//--- Generated by OneClick Automation SourceGenerator v.3.0 ---
DATA_BLOCK DB111
TITLE =Sensors 4-20
AUTHOR:  Kratovi4
VERSION : 2.0
STRUCT
SNS: ARRAY  [1 .. 25] OF
"SNS"; // Array
END_STRUCT ;
BEGIN
END_DATA_BLOCK


DATA_BLOCK DB121
TITLE =Sensors 4-20
AUTHOR:  Kratovi4
VERSION : 2.0
STRUCT
SNS: ARRAY  [1 .. 30] OF
"SNS"; // Array
END_STRUCT ;
BEGIN
END_DATA_BLOCK


DATA_BLOCK DB131
TITLE =Sensors 4-20
AUTHOR:  Kratovi4
VERSION : 2.0
STRUCT
SNS: ARRAY  [1 .. 5] OF
"SNS"; // Array
END_STRUCT ;
BEGIN
END_DATA_BLOCK


DATA_BLOCK DB141
TITLE =Sensors 4-20
AUTHOR:  Kratovi4
VERSION : 2.0
STRUCT
SNS: ARRAY  [1 .. 5] OF
"SNS"; // Array
END_STRUCT ;
BEGIN
END_DATA_BLOCK


DATA_BLOCK DB151
TITLE =Sensors 4-20
AUTHOR:  Kratovi4
VERSION : 2.0
STRUCT
SNS: ARRAY  [1 .. 5] OF
"SNS"; // Array
END_STRUCT ;
BEGIN
END_DATA_BLOCK


DATA_BLOCK DB161
TITLE =Sensors 4-20
AUTHOR:  Kratovi4
VERSION : 2.0
STRUCT
SNS: ARRAY  [1 .. 5] OF
"SNS"; // Array
END_STRUCT ;
BEGIN
END_DATA_BLOCK


DATA_BLOCK DB171
TITLE =Sensors 4-20
AUTHOR:  Kratovi4
VERSION : 2.0
STRUCT
SNS: ARRAY  [1 .. 5] OF
"SNS"; // Array
END_STRUCT ;
BEGIN
END_DATA_BLOCK


DATA_BLOCK DB211
TITLE =Sensors 4-20
AUTHOR:  Kratovi4
VERSION : 2.0
STRUCT
SNS: ARRAY  [1 .. 10] OF
"SNS"; // Array
END_STRUCT ;
BEGIN
END_DATA_BLOCK


DATA_BLOCK DB221
TITLE =Sensors 4-20
AUTHOR:  Kratovi4
VERSION : 2.0
STRUCT
SNS: ARRAY  [1 .. 10] OF
"SNS"; // Array
END_STRUCT ;
BEGIN
END_DATA_BLOCK


DATA_BLOCK DB231
TITLE =Sensors 4-20
AUTHOR:  Kratovi4
VERSION : 2.0
STRUCT
SNS: ARRAY  [1 .. 10] OF
"SNS"; // Array
END_STRUCT ;
BEGIN
END_DATA_BLOCK


DATA_BLOCK DB241
TITLE =Sensors 4-20
AUTHOR:  Kratovi4
VERSION : 2.0
STRUCT
SNS: ARRAY  [1 .. 5] OF
"SNS"; // Array
END_STRUCT ;
BEGIN
END_DATA_BLOCK


DATA_BLOCK DB251
TITLE =Sensors 4-20
AUTHOR:  Kratovi4
VERSION : 2.0
STRUCT
SNS: ARRAY  [1 .. 5] OF
"SNS"; // Array
END_STRUCT ;
BEGIN
END_DATA_BLOCK


DATA_BLOCK DB261
TITLE =Sensors 4-20
AUTHOR:  Kratovi4
VERSION : 2.0
STRUCT
SNS: ARRAY  [1 .. 5] OF
"SNS"; // Array
END_STRUCT ;
BEGIN
END_DATA_BLOCK


DATA_BLOCK DB291
TITLE =Sensors 4-20
AUTHOR:  Kratovi4
VERSION : 2.0
STRUCT
SNS: ARRAY  [1 .. 25] OF
"SNS"; // Array
END_STRUCT ;
BEGIN
END_DATA_BLOCK


DATA_BLOCK DB301
TITLE =Sensors 4-20
AUTHOR:  Kratovi4
VERSION : 2.0
STRUCT
SNS: ARRAY  [1 .. 10] OF
"SNS"; // Array
END_STRUCT ;
BEGIN
END_DATA_BLOCK


DATA_BLOCK DB311
TITLE =Sensors 4-20
AUTHOR:  Kratovi4
VERSION : 2.0
STRUCT
SNS: ARRAY  [1 .. 5] OF
"SNS"; // Array
END_STRUCT ;
BEGIN
END_DATA_BLOCK


DATA_BLOCK DB321
TITLE =Sensors 4-20
AUTHOR:  Kratovi4
VERSION : 2.0
STRUCT
SNS: ARRAY  [1 .. 5] OF
"SNS"; // Array
END_STRUCT ;
BEGIN
END_DATA_BLOCK


DATA_BLOCK DB341
TITLE =Sensors 4-20
AUTHOR:  Kratovi4
VERSION : 2.0
STRUCT
SNS: ARRAY  [1 .. 5] OF
"SNS"; // Array
END_STRUCT ;
BEGIN
END_DATA_BLOCK


DATA_BLOCK DB431
TITLE =Sensors 4-20
AUTHOR:  Kratovi4
VERSION : 2.0
STRUCT
SNS: ARRAY  [1 .. 20] OF
"SNS"; // Array
END_STRUCT ;
BEGIN
END_DATA_BLOCK


DATA_BLOCK DB441
TITLE =Sensors 4-20
AUTHOR:  Kratovi4
VERSION : 2.0
STRUCT
SNS: ARRAY  [1 .. 5] OF
"SNS"; // Array
END_STRUCT ;
BEGIN
END_DATA_BLOCK


DATA_BLOCK DB451
TITLE =Sensors 4-20
AUTHOR:  Kratovi4
VERSION : 2.0
STRUCT
SNS: ARRAY  [1 .. 5] OF
"SNS"; // Array
END_STRUCT ;
BEGIN
END_DATA_BLOCK


DATA_BLOCK DB461
TITLE =Sensors 4-20
AUTHOR:  Kratovi4
VERSION : 2.0
STRUCT
SNS: ARRAY  [1 .. 5] OF
"SNS"; // Array
END_STRUCT ;
BEGIN
END_DATA_BLOCK


DATA_BLOCK DB471
TITLE =Sensors 4-20
AUTHOR:  Kratovi4
VERSION : 2.0
STRUCT
SNS: ARRAY  [1 .. 5] OF
"SNS"; // Array
END_STRUCT ;
BEGIN
END_DATA_BLOCK


DATA_BLOCK DB511
TITLE =Sensors 4-20
AUTHOR:  Kratovi4
VERSION : 2.0
STRUCT
SNS: ARRAY  [1 .. 5] OF
"SNS"; // Array
END_STRUCT ;
BEGIN
END_DATA_BLOCK


DATA_BLOCK DB521
TITLE =Sensors 4-20
AUTHOR:  Kratovi4
VERSION : 2.0
STRUCT
SNS: ARRAY  [1 .. 5] OF
"SNS"; // Array
END_STRUCT ;
BEGIN
END_DATA_BLOCK


DATA_BLOCK DB531
TITLE =Sensors 4-20
AUTHOR:  Kratovi4
VERSION : 2.0
STRUCT
SNS: ARRAY  [1 .. 5] OF
"SNS"; // Array
END_STRUCT ;
BEGIN
END_DATA_BLOCK


DATA_BLOCK DB541
TITLE =Sensors 4-20
AUTHOR:  Kratovi4
VERSION : 2.0
STRUCT
SNS: ARRAY  [1 .. 5] OF
"SNS"; // Array
END_STRUCT ;
BEGIN
END_DATA_BLOCK


DATA_BLOCK DB561
TITLE =Sensors 4-20
AUTHOR:  Kratovi4
VERSION : 2.0
STRUCT
SNS: ARRAY  [1 .. 5] OF
"SNS"; // Array
END_STRUCT ;
BEGIN
END_DATA_BLOCK


DATA_BLOCK DB571
TITLE =Sensors 4-20
AUTHOR:  Kratovi4
VERSION : 2.0
STRUCT
SNS: ARRAY  [1 .. 5] OF
"SNS"; // Array
END_STRUCT ;
BEGIN
END_DATA_BLOCK


DATA_BLOCK DB581
TITLE =Sensors 4-20
AUTHOR:  Kratovi4
VERSION : 2.0
STRUCT
SNS: ARRAY  [1 .. 5] OF
"SNS"; // Array
END_STRUCT ;
BEGIN
END_DATA_BLOCK


DATA_BLOCK DB611
TITLE =Sensors 4-20
AUTHOR:  Kratovi4
VERSION : 2.0
STRUCT
SNS: ARRAY  [1 .. 5] OF
"SNS"; // Array
END_STRUCT ;
BEGIN
END_DATA_BLOCK


DATA_BLOCK DB671
TITLE =Sensors 4-20
AUTHOR:  Kratovi4
VERSION : 2.0
STRUCT
SNS: ARRAY  [1 .. 10] OF
"SNS"; // Array
END_STRUCT ;
BEGIN
END_DATA_BLOCK


DATA_BLOCK DB681
TITLE =Sensors 4-20
AUTHOR:  Kratovi4
VERSION : 2.0
STRUCT
SNS: ARRAY  [1 .. 5] OF
"SNS"; // Array
END_STRUCT ;
BEGIN
END_DATA_BLOCK


DATA_BLOCK DB691
TITLE =Sensors 4-20
AUTHOR:  Kratovi4
VERSION : 2.0
STRUCT
SNS: ARRAY  [1 .. 5] OF
"SNS"; // Array
END_STRUCT ;
BEGIN
END_DATA_BLOCK


DATA_BLOCK DB701
TITLE =Sensors 4-20
AUTHOR:  Kratovi4
VERSION : 2.0
STRUCT
SNS: ARRAY  [1 .. 5] OF
"SNS"; // Array
END_STRUCT ;
BEGIN
END_DATA_BLOCK


DATA_BLOCK DB711
TITLE =Sensors 4-20
AUTHOR:  Kratovi4
VERSION : 2.0
STRUCT
SNS: ARRAY  [1 .. 5] OF
"SNS"; // Array
END_STRUCT ;
BEGIN
END_DATA_BLOCK


DATA_BLOCK DB721
TITLE =Sensors 4-20
AUTHOR:  Kratovi4
VERSION : 2.0
STRUCT
SNS: ARRAY  [1 .. 15] OF
"SNS"; // Array
END_STRUCT ;
BEGIN
END_DATA_BLOCK


DATA_BLOCK DB731
TITLE =Sensors 4-20
AUTHOR:  Kratovi4
VERSION : 2.0
STRUCT
SNS: ARRAY  [1 .. 5] OF
"SNS"; // Array
END_STRUCT ;
BEGIN
END_DATA_BLOCK


DATA_BLOCK DB741
TITLE =Sensors 4-20
AUTHOR:  Kratovi4
VERSION : 2.0
STRUCT
SNS: ARRAY  [1 .. 5] OF
"SNS"; // Array
END_STRUCT ;
BEGIN
END_DATA_BLOCK


DATA_BLOCK DB751
TITLE =Sensors 4-20
AUTHOR:  Kratovi4
VERSION : 2.0
STRUCT
SNS: ARRAY  [1 .. 5] OF
"SNS"; // Array
END_STRUCT ;
BEGIN
END_DATA_BLOCK


DATA_BLOCK DB771
TITLE =Sensors 4-20
AUTHOR:  Kratovi4
VERSION : 2.0
STRUCT
SNS: ARRAY  [1 .. 5] OF
"SNS"; // Array
END_STRUCT ;
BEGIN
END_DATA_BLOCK


DATA_BLOCK DB781
TITLE =Sensors 4-20
AUTHOR:  Kratovi4
VERSION : 2.0
STRUCT
SNS: ARRAY  [1 .. 5] OF
"SNS"; // Array
END_STRUCT ;
BEGIN
END_DATA_BLOCK


DATA_BLOCK DB791
TITLE =Sensors 4-20
AUTHOR:  Kratovi4
VERSION : 2.0
STRUCT
SNS: ARRAY  [1 .. 5] OF
"SNS"; // Array
END_STRUCT ;
BEGIN
END_DATA_BLOCK


DATA_BLOCK DB801
TITLE =Sensors 4-20
AUTHOR:  Kratovi4
VERSION : 2.0
STRUCT
SNS: ARRAY  [1 .. 5] OF
"SNS"; // Array
END_STRUCT ;
BEGIN
END_DATA_BLOCK


DATA_BLOCK DB811
TITLE =Sensors 4-20
AUTHOR:  Kratovi4
VERSION : 2.0
STRUCT
SNS: ARRAY  [1 .. 5] OF
"SNS"; // Array
END_STRUCT ;
BEGIN
END_DATA_BLOCK


DATA_BLOCK DB831
TITLE =Sensors 4-20
AUTHOR:  Kratovi4
VERSION : 2.0
STRUCT
SNS: ARRAY  [1 .. 5] OF
"SNS"; // Array
END_STRUCT ;
BEGIN
END_DATA_BLOCK


DATA_BLOCK DB841
TITLE =Sensors 4-20
AUTHOR:  Kratovi4
VERSION : 2.0
STRUCT
SNS: ARRAY  [1 .. 5] OF
"SNS"; // Array
END_STRUCT ;
BEGIN
END_DATA_BLOCK


DATA_BLOCK DB851
TITLE =Sensors 4-20
AUTHOR:  Kratovi4
VERSION : 2.0
STRUCT
SNS: ARRAY  [1 .. 5] OF
"SNS"; // Array
END_STRUCT ;
BEGIN
END_DATA_BLOCK


DATA_BLOCK DB861
TITLE =Sensors 4-20
AUTHOR:  Kratovi4
VERSION : 2.0
STRUCT
SNS: ARRAY  [1 .. 5] OF
"SNS"; // Array
END_STRUCT ;
BEGIN
END_DATA_BLOCK


DATA_BLOCK DB881
TITLE =Sensors 4-20
AUTHOR:  Kratovi4
VERSION : 2.0
STRUCT
SNS: ARRAY  [1 .. 5] OF
"SNS"; // Array
END_STRUCT ;
BEGIN
END_DATA_BLOCK


DATA_BLOCK DB122
TITLE =Discrette signals
AUTHOR:  Kratovi4
VERSION : 2.0
STRUCT
SNB: ARRAY  [1 .. 55] OF
"SND"; // Array
END_STRUCT ;
BEGIN
END_DATA_BLOCK


DATA_BLOCK DB142
TITLE =Discrette signals
AUTHOR:  Kratovi4
VERSION : 2.0
STRUCT
SNB: ARRAY  [1 .. 55] OF
"SND"; // Array
END_STRUCT ;
BEGIN
END_DATA_BLOCK


DATA_BLOCK DB162
TITLE =Discrette signals
AUTHOR:  Kratovi4
VERSION : 2.0
STRUCT
SNB: ARRAY  [1 .. 55] OF
"SND"; // Array
END_STRUCT ;
BEGIN
END_DATA_BLOCK


DATA_BLOCK DB172
TITLE =Discrette signals
AUTHOR:  Kratovi4
VERSION : 2.0
STRUCT
SNB: ARRAY  [1 .. 55] OF
"SND"; // Array
END_STRUCT ;
BEGIN
END_DATA_BLOCK


DATA_BLOCK DB242
TITLE =Discrette signals
AUTHOR:  Kratovi4
VERSION : 2.0
STRUCT
SNB: ARRAY  [1 .. 55] OF
"SND"; // Array
END_STRUCT ;
BEGIN
END_DATA_BLOCK


DATA_BLOCK DB252
TITLE =Discrette signals
AUTHOR:  Kratovi4
VERSION : 2.0
STRUCT
SNB: ARRAY  [1 .. 55] OF
"SND"; // Array
END_STRUCT ;
BEGIN
END_DATA_BLOCK


DATA_BLOCK DB262
TITLE =Discrette signals
AUTHOR:  Kratovi4
VERSION : 2.0
STRUCT
SNB: ARRAY  [1 .. 55] OF
"SND"; // Array
END_STRUCT ;
BEGIN
END_DATA_BLOCK


DATA_BLOCK DB312
TITLE =Discrette signals
AUTHOR:  Kratovi4
VERSION : 2.0
STRUCT
SNB: ARRAY  [1 .. 55] OF
"SND"; // Array
END_STRUCT ;
BEGIN
END_DATA_BLOCK


DATA_BLOCK DB322
TITLE =Discrette signals
AUTHOR:  Kratovi4
VERSION : 2.0
STRUCT
SNB: ARRAY  [1 .. 55] OF
"SND"; // Array
END_STRUCT ;
BEGIN
END_DATA_BLOCK


DATA_BLOCK DB442
TITLE =Discrette signals
AUTHOR:  Kratovi4
VERSION : 2.0
STRUCT
SNB: ARRAY  [1 .. 55] OF
"SND"; // Array
END_STRUCT ;
BEGIN
END_DATA_BLOCK


DATA_BLOCK DB452
TITLE =Discrette signals
AUTHOR:  Kratovi4
VERSION : 2.0
STRUCT
SNB: ARRAY  [1 .. 55] OF
"SND"; // Array
END_STRUCT ;
BEGIN
END_DATA_BLOCK


DATA_BLOCK DB462
TITLE =Discrette signals
AUTHOR:  Kratovi4
VERSION : 2.0
STRUCT
SNB: ARRAY  [1 .. 55] OF
"SND"; // Array
END_STRUCT ;
BEGIN
END_DATA_BLOCK


DATA_BLOCK DB472
TITLE =Discrette signals
AUTHOR:  Kratovi4
VERSION : 2.0
STRUCT
SNB: ARRAY  [1 .. 55] OF
"SND"; // Array
END_STRUCT ;
BEGIN
END_DATA_BLOCK


DATA_BLOCK DB522
TITLE =Discrette signals
AUTHOR:  Kratovi4
VERSION : 2.0
STRUCT
SNB: ARRAY  [1 .. 55] OF
"SND"; // Array
END_STRUCT ;
BEGIN
END_DATA_BLOCK


DATA_BLOCK DB532
TITLE =Discrette signals
AUTHOR:  Kratovi4
VERSION : 2.0
STRUCT
SNB: ARRAY  [1 .. 55] OF
"SND"; // Array
END_STRUCT ;
BEGIN
END_DATA_BLOCK


DATA_BLOCK DB562
TITLE =Discrette signals
AUTHOR:  Kratovi4
VERSION : 2.0
STRUCT
SNB: ARRAY  [1 .. 60] OF
"SND"; // Array
END_STRUCT ;
BEGIN
END_DATA_BLOCK


DATA_BLOCK DB572
TITLE =Discrette signals
AUTHOR:  Kratovi4
VERSION : 2.0
STRUCT
SNB: ARRAY  [1 .. 60] OF
"SND"; // Array
END_STRUCT ;
BEGIN
END_DATA_BLOCK


DATA_BLOCK DB582
TITLE =Discrette signals
AUTHOR:  Kratovi4
VERSION : 2.0
STRUCT
SNB: ARRAY  [1 .. 60] OF
"SND"; // Array
END_STRUCT ;
BEGIN
END_DATA_BLOCK


DATA_BLOCK DB602
TITLE =Discrette signals
AUTHOR:  Kratovi4
VERSION : 2.0
STRUCT
SNB: ARRAY  [1 .. 10] OF
"SND"; // Array
END_STRUCT ;
BEGIN
END_DATA_BLOCK


DATA_BLOCK DB682
TITLE =Discrette signals
AUTHOR:  Kratovi4
VERSION : 2.0
STRUCT
SNB: ARRAY  [1 .. 55] OF
"SND"; // Array
END_STRUCT ;
BEGIN
END_DATA_BLOCK


DATA_BLOCK DB692
TITLE =Discrette signals
AUTHOR:  Kratovi4
VERSION : 2.0
STRUCT
SNB: ARRAY  [1 .. 55] OF
"SND"; // Array
END_STRUCT ;
BEGIN
END_DATA_BLOCK


DATA_BLOCK DB702
TITLE =Discrette signals
AUTHOR:  Kratovi4
VERSION : 2.0
STRUCT
SNB: ARRAY  [1 .. 55] OF
"SND"; // Array
END_STRUCT ;
BEGIN
END_DATA_BLOCK


DATA_BLOCK DB712
TITLE =Discrette signals
AUTHOR:  Kratovi4
VERSION : 2.0
STRUCT
SNB: ARRAY  [1 .. 55] OF
"SND"; // Array
END_STRUCT ;
BEGIN
END_DATA_BLOCK


DATA_BLOCK DB732
TITLE =Discrette signals
AUTHOR:  Kratovi4
VERSION : 2.0
STRUCT
SNB: ARRAY  [1 .. 55] OF
"SND"; // Array
END_STRUCT ;
BEGIN
END_DATA_BLOCK


DATA_BLOCK DB742
TITLE =Discrette signals
AUTHOR:  Kratovi4
VERSION : 2.0
STRUCT
SNB: ARRAY  [1 .. 55] OF
"SND"; // Array
END_STRUCT ;
BEGIN
END_DATA_BLOCK


DATA_BLOCK DB752
TITLE =Discrette signals
AUTHOR:  Kratovi4
VERSION : 2.0
STRUCT
SNB: ARRAY  [1 .. 55] OF
"SND"; // Array
END_STRUCT ;
BEGIN
END_DATA_BLOCK


DATA_BLOCK DB792
TITLE =Discrette signals
AUTHOR:  Kratovi4
VERSION : 2.0
STRUCT
SNB: ARRAY  [1 .. 55] OF
"SND"; // Array
END_STRUCT ;
BEGIN
END_DATA_BLOCK


DATA_BLOCK DB802
TITLE =Discrette signals
AUTHOR:  Kratovi4
VERSION : 2.0
STRUCT
SNB: ARRAY  [1 .. 55] OF
"SND"; // Array
END_STRUCT ;
BEGIN
END_DATA_BLOCK


DATA_BLOCK DB832
TITLE =Discrette signals
AUTHOR:  Kratovi4
VERSION : 2.0
STRUCT
SNB: ARRAY  [1 .. 55] OF
"SND"; // Array
END_STRUCT ;
BEGIN
END_DATA_BLOCK


DATA_BLOCK DB842
TITLE =Discrette signals
AUTHOR:  Kratovi4
VERSION : 2.0
STRUCT
SNB: ARRAY  [1 .. 55] OF
"SND"; // Array
END_STRUCT ;
BEGIN
END_DATA_BLOCK


DATA_BLOCK DB852
TITLE =Discrette signals
AUTHOR:  Kratovi4
VERSION : 2.0
STRUCT
SNB: ARRAY  [1 .. 55] OF
"SND"; // Array
END_STRUCT ;
BEGIN
END_DATA_BLOCK


DATA_BLOCK DB862
TITLE =Discrette signals
AUTHOR:  Kratovi4
VERSION : 2.0
STRUCT
SNB: ARRAY  [1 .. 55] OF
"SND"; // Array
END_STRUCT ;
BEGIN
END_DATA_BLOCK


DATA_BLOCK DB882
TITLE =Discrette signals
AUTHOR:  Kratovi4
VERSION : 2.0
STRUCT
SNB: ARRAY  [1 .. 55] OF
"SND"; // Array
END_STRUCT ;
BEGIN
END_DATA_BLOCK


DATA_BLOCK DB113
TITLE =Level sensors
AUTHOR:  Kratovi4
VERSION : 2.0
STRUCT
SND: ARRAY  [1 .. 20] OF
"SND"; // Array
END_STRUCT ;
BEGIN
END_DATA_BLOCK


DATA_BLOCK DB123
TITLE =Level sensors
AUTHOR:  Kratovi4
VERSION : 2.0
STRUCT
SND: ARRAY  [1 .. 25] OF
"SND"; // Array
END_STRUCT ;
BEGIN
END_DATA_BLOCK


DATA_BLOCK DB133
TITLE =Level sensors
AUTHOR:  Kratovi4
VERSION : 2.0
STRUCT
SND: ARRAY  [1 .. 5] OF
"SND"; // Array
END_STRUCT ;
BEGIN
END_DATA_BLOCK


DATA_BLOCK DB143
TITLE =Level sensors
AUTHOR:  Kratovi4
VERSION : 2.0
STRUCT
SND: ARRAY  [1 .. 5] OF
"SND"; // Array
END_STRUCT ;
BEGIN
END_DATA_BLOCK


DATA_BLOCK DB153
TITLE =Level sensors
AUTHOR:  Kratovi4
VERSION : 2.0
STRUCT
SND: ARRAY  [1 .. 5] OF
"SND"; // Array
END_STRUCT ;
BEGIN
END_DATA_BLOCK


DATA_BLOCK DB163
TITLE =Level sensors
AUTHOR:  Kratovi4
VERSION : 2.0
STRUCT
SND: ARRAY  [1 .. 5] OF
"SND"; // Array
END_STRUCT ;
BEGIN
END_DATA_BLOCK


DATA_BLOCK DB173
TITLE =Level sensors
AUTHOR:  Kratovi4
VERSION : 2.0
STRUCT
SND: ARRAY  [1 .. 5] OF
"SND"; // Array
END_STRUCT ;
BEGIN
END_DATA_BLOCK


DATA_BLOCK DB213
TITLE =Level sensors
AUTHOR:  Kratovi4
VERSION : 2.0
STRUCT
SND: ARRAY  [1 .. 5] OF
"SND"; // Array
END_STRUCT ;
BEGIN
END_DATA_BLOCK


DATA_BLOCK DB223
TITLE =Level sensors
AUTHOR:  Kratovi4
VERSION : 2.0
STRUCT
SND: ARRAY  [1 .. 5] OF
"SND"; // Array
END_STRUCT ;
BEGIN
END_DATA_BLOCK


DATA_BLOCK DB233
TITLE =Level sensors
AUTHOR:  Kratovi4
VERSION : 2.0
STRUCT
SND: ARRAY  [1 .. 5] OF
"SND"; // Array
END_STRUCT ;
BEGIN
END_DATA_BLOCK


DATA_BLOCK DB243
TITLE =Level sensors
AUTHOR:  Kratovi4
VERSION : 2.0
STRUCT
SND: ARRAY  [1 .. 5] OF
"SND"; // Array
END_STRUCT ;
BEGIN
END_DATA_BLOCK


DATA_BLOCK DB253
TITLE =Level sensors
AUTHOR:  Kratovi4
VERSION : 2.0
STRUCT
SND: ARRAY  [1 .. 5] OF
"SND"; // Array
END_STRUCT ;
BEGIN
END_DATA_BLOCK


DATA_BLOCK DB263
TITLE =Level sensors
AUTHOR:  Kratovi4
VERSION : 2.0
STRUCT
SND: ARRAY  [1 .. 5] OF
"SND"; // Array
END_STRUCT ;
BEGIN
END_DATA_BLOCK


DATA_BLOCK DB293
TITLE =Level sensors
AUTHOR:  Kratovi4
VERSION : 2.0
STRUCT
SND: ARRAY  [1 .. 15] OF
"SND"; // Array
END_STRUCT ;
BEGIN
END_DATA_BLOCK


DATA_BLOCK DB303
TITLE =Level sensors
AUTHOR:  Kratovi4
VERSION : 2.0
STRUCT
SND: ARRAY  [1 .. 5] OF
"SND"; // Array
END_STRUCT ;
BEGIN
END_DATA_BLOCK


DATA_BLOCK DB313
TITLE =Level sensors
AUTHOR:  Kratovi4
VERSION : 2.0
STRUCT
SND: ARRAY  [1 .. 5] OF
"SND"; // Array
END_STRUCT ;
BEGIN
END_DATA_BLOCK


DATA_BLOCK DB323
TITLE =Level sensors
AUTHOR:  Kratovi4
VERSION : 2.0
STRUCT
SND: ARRAY  [1 .. 5] OF
"SND"; // Array
END_STRUCT ;
BEGIN
END_DATA_BLOCK


DATA_BLOCK DB433
TITLE =Level sensors
AUTHOR:  Kratovi4
VERSION : 2.0
STRUCT
SND: ARRAY  [1 .. 25] OF
"SND"; // Array
END_STRUCT ;
BEGIN
END_DATA_BLOCK


DATA_BLOCK DB443
TITLE =Level sensors
AUTHOR:  Kratovi4
VERSION : 2.0
STRUCT
SND: ARRAY  [1 .. 5] OF
"SND"; // Array
END_STRUCT ;
BEGIN
END_DATA_BLOCK


DATA_BLOCK DB453
TITLE =Level sensors
AUTHOR:  Kratovi4
VERSION : 2.0
STRUCT
SND: ARRAY  [1 .. 5] OF
"SND"; // Array
END_STRUCT ;
BEGIN
END_DATA_BLOCK


DATA_BLOCK DB463
TITLE =Level sensors
AUTHOR:  Kratovi4
VERSION : 2.0
STRUCT
SND: ARRAY  [1 .. 5] OF
"SND"; // Array
END_STRUCT ;
BEGIN
END_DATA_BLOCK


DATA_BLOCK DB473
TITLE =Level sensors
AUTHOR:  Kratovi4
VERSION : 2.0
STRUCT
SND: ARRAY  [1 .. 5] OF
"SND"; // Array
END_STRUCT ;
BEGIN
END_DATA_BLOCK


DATA_BLOCK DB523
TITLE =Level sensors
AUTHOR:  Kratovi4
VERSION : 2.0
STRUCT
SND: ARRAY  [1 .. 5] OF
"SND"; // Array
END_STRUCT ;
BEGIN
END_DATA_BLOCK


DATA_BLOCK DB533
TITLE =Level sensors
AUTHOR:  Kratovi4
VERSION : 2.0
STRUCT
SND: ARRAY  [1 .. 5] OF
"SND"; // Array
END_STRUCT ;
BEGIN
END_DATA_BLOCK


DATA_BLOCK DB553
TITLE =Level sensors
AUTHOR:  Kratovi4
VERSION : 2.0
STRUCT
SND: ARRAY  [1 .. 5] OF
"SND"; // Array
END_STRUCT ;
BEGIN
END_DATA_BLOCK


DATA_BLOCK DB563
TITLE =Level sensors
AUTHOR:  Kratovi4
VERSION : 2.0
STRUCT
SND: ARRAY  [1 .. 5] OF
"SND"; // Array
END_STRUCT ;
BEGIN
END_DATA_BLOCK


DATA_BLOCK DB573
TITLE =Level sensors
AUTHOR:  Kratovi4
VERSION : 2.0
STRUCT
SND: ARRAY  [1 .. 5] OF
"SND"; // Array
END_STRUCT ;
BEGIN
END_DATA_BLOCK


DATA_BLOCK DB583
TITLE =Level sensors
AUTHOR:  Kratovi4
VERSION : 2.0
STRUCT
SND: ARRAY  [1 .. 5] OF
"SND"; // Array
END_STRUCT ;
BEGIN
END_DATA_BLOCK


DATA_BLOCK DB603
TITLE =Level sensors
AUTHOR:  Kratovi4
VERSION : 2.0
STRUCT
SND: ARRAY  [1 .. 5] OF
"SND"; // Array
END_STRUCT ;
BEGIN
END_DATA_BLOCK


DATA_BLOCK DB673
TITLE =Level sensors
AUTHOR:  Kratovi4
VERSION : 2.0
STRUCT
SND: ARRAY  [1 .. 5] OF
"SND"; // Array
END_STRUCT ;
BEGIN
END_DATA_BLOCK


DATA_BLOCK DB683
TITLE =Level sensors
AUTHOR:  Kratovi4
VERSION : 2.0
STRUCT
SND: ARRAY  [1 .. 5] OF
"SND"; // Array
END_STRUCT ;
BEGIN
END_DATA_BLOCK


DATA_BLOCK DB693
TITLE =Level sensors
AUTHOR:  Kratovi4
VERSION : 2.0
STRUCT
SND: ARRAY  [1 .. 5] OF
"SND"; // Array
END_STRUCT ;
BEGIN
END_DATA_BLOCK


DATA_BLOCK DB703
TITLE =Level sensors
AUTHOR:  Kratovi4
VERSION : 2.0
STRUCT
SND: ARRAY  [1 .. 5] OF
"SND"; // Array
END_STRUCT ;
BEGIN
END_DATA_BLOCK


DATA_BLOCK DB713
TITLE =Level sensors
AUTHOR:  Kratovi4
VERSION : 2.0
STRUCT
SND: ARRAY  [1 .. 5] OF
"SND"; // Array
END_STRUCT ;
BEGIN
END_DATA_BLOCK


DATA_BLOCK DB723
TITLE =Level sensors
AUTHOR:  Kratovi4
VERSION : 2.0
STRUCT
SND: ARRAY  [1 .. 15] OF
"SND"; // Array
END_STRUCT ;
BEGIN
END_DATA_BLOCK


DATA_BLOCK DB733
TITLE =Level sensors
AUTHOR:  Kratovi4
VERSION : 2.0
STRUCT
SND: ARRAY  [1 .. 5] OF
"SND"; // Array
END_STRUCT ;
BEGIN
END_DATA_BLOCK


DATA_BLOCK DB743
TITLE =Level sensors
AUTHOR:  Kratovi4
VERSION : 2.0
STRUCT
SND: ARRAY  [1 .. 5] OF
"SND"; // Array
END_STRUCT ;
BEGIN
END_DATA_BLOCK


DATA_BLOCK DB753
TITLE =Level sensors
AUTHOR:  Kratovi4
VERSION : 2.0
STRUCT
SND: ARRAY  [1 .. 5] OF
"SND"; // Array
END_STRUCT ;
BEGIN
END_DATA_BLOCK


DATA_BLOCK DB793
TITLE =Level sensors
AUTHOR:  Kratovi4
VERSION : 2.0
STRUCT
SND: ARRAY  [1 .. 5] OF
"SND"; // Array
END_STRUCT ;
BEGIN
END_DATA_BLOCK


DATA_BLOCK DB803
TITLE =Level sensors
AUTHOR:  Kratovi4
VERSION : 2.0
STRUCT
SND: ARRAY  [1 .. 5] OF
"SND"; // Array
END_STRUCT ;
BEGIN
END_DATA_BLOCK


DATA_BLOCK DB833
TITLE =Level sensors
AUTHOR:  Kratovi4
VERSION : 2.0
STRUCT
SND: ARRAY  [1 .. 5] OF
"SND"; // Array
END_STRUCT ;
BEGIN
END_DATA_BLOCK


DATA_BLOCK DB843
TITLE =Level sensors
AUTHOR:  Kratovi4
VERSION : 2.0
STRUCT
SND: ARRAY  [1 .. 5] OF
"SND"; // Array
END_STRUCT ;
BEGIN
END_DATA_BLOCK


DATA_BLOCK DB853
TITLE =Level sensors
AUTHOR:  Kratovi4
VERSION : 2.0
STRUCT
SND: ARRAY  [1 .. 5] OF
"SND"; // Array
END_STRUCT ;
BEGIN
END_DATA_BLOCK


DATA_BLOCK DB863
TITLE =Level sensors
AUTHOR:  Kratovi4
VERSION : 2.0
STRUCT
SND: ARRAY  [1 .. 5] OF
"SND"; // Array
END_STRUCT ;
BEGIN
END_DATA_BLOCK


DATA_BLOCK DB883
TITLE =Level sensors
AUTHOR:  Kratovi4
VERSION : 2.0
STRUCT
SND: ARRAY  [1 .. 10] OF
"SND"; // Array
END_STRUCT ;
BEGIN
END_DATA_BLOCK


DATA_BLOCK DB114
TITLE =Valves
AUTHOR:  Kratovi4
VERSION : 2.0
STRUCT
DRV: ARRAY  [1 .. 55] OF
"DRV"; // Array
END_STRUCT ;
BEGIN
END_DATA_BLOCK


DATA_BLOCK DB124
TITLE =Valves
AUTHOR:  Kratovi4
VERSION : 2.0
STRUCT
DRV: ARRAY  [1 .. 80] OF
"DRV"; // Array
END_STRUCT ;
BEGIN
END_DATA_BLOCK


DATA_BLOCK DB134
TITLE =Valves
AUTHOR:  Kratovi4
VERSION : 2.0
STRUCT
DRV: ARRAY  [1 .. 5] OF
"DRV"; // Array
END_STRUCT ;
BEGIN
END_DATA_BLOCK


DATA_BLOCK DB144
TITLE =Valves
AUTHOR:  Kratovi4
VERSION : 2.0
STRUCT
DRV: ARRAY  [1 .. 5] OF
"DRV"; // Array
END_STRUCT ;
BEGIN
END_DATA_BLOCK


DATA_BLOCK DB154
TITLE =Valves
AUTHOR:  Kratovi4
VERSION : 2.0
STRUCT
DRV: ARRAY  [1 .. 5] OF
"DRV"; // Array
END_STRUCT ;
BEGIN
END_DATA_BLOCK


DATA_BLOCK DB164
TITLE =Valves
AUTHOR:  Kratovi4
VERSION : 2.0
STRUCT
DRV: ARRAY  [1 .. 5] OF
"DRV"; // Array
END_STRUCT ;
BEGIN
END_DATA_BLOCK


DATA_BLOCK DB174
TITLE =Valves
AUTHOR:  Kratovi4
VERSION : 2.0
STRUCT
DRV: ARRAY  [1 .. 5] OF
"DRV"; // Array
END_STRUCT ;
BEGIN
END_DATA_BLOCK


DATA_BLOCK DB204
TITLE =Valves
AUTHOR:  Kratovi4
VERSION : 2.0
STRUCT
DRV: ARRAY  [1 .. 5] OF
"DRV"; // Array
END_STRUCT ;
BEGIN
END_DATA_BLOCK


DATA_BLOCK DB214
TITLE =Valves
AUTHOR:  Kratovi4
VERSION : 2.0
STRUCT
DRV: ARRAY  [1 .. 10] OF
"DRV"; // Array
END_STRUCT ;
BEGIN
END_DATA_BLOCK


DATA_BLOCK DB224
TITLE =Valves
AUTHOR:  Kratovi4
VERSION : 2.0
STRUCT
DRV: ARRAY  [1 .. 10] OF
"DRV"; // Array
END_STRUCT ;
BEGIN
END_DATA_BLOCK


DATA_BLOCK DB234
TITLE =Valves
AUTHOR:  Kratovi4
VERSION : 2.0
STRUCT
DRV: ARRAY  [1 .. 10] OF
"DRV"; // Array
END_STRUCT ;
BEGIN
END_DATA_BLOCK


DATA_BLOCK DB244
TITLE =Valves
AUTHOR:  Kratovi4
VERSION : 2.0
STRUCT
DRV: ARRAY  [1 .. 10] OF
"DRV"; // Array
END_STRUCT ;
BEGIN
END_DATA_BLOCK


DATA_BLOCK DB254
TITLE =Valves
AUTHOR:  Kratovi4
VERSION : 2.0
STRUCT
DRV: ARRAY  [1 .. 10] OF
"DRV"; // Array
END_STRUCT ;
BEGIN
END_DATA_BLOCK


DATA_BLOCK DB264
TITLE =Valves
AUTHOR:  Kratovi4
VERSION : 2.0
STRUCT
DRV: ARRAY  [1 .. 10] OF
"DRV"; // Array
END_STRUCT ;
BEGIN
END_DATA_BLOCK


DATA_BLOCK DB284
TITLE =Valves
AUTHOR:  Kratovi4
VERSION : 2.0
STRUCT
DRV: ARRAY  [1 .. 5] OF
"DRV"; // Array
END_STRUCT ;
BEGIN
END_DATA_BLOCK


DATA_BLOCK DB294
TITLE =Valves
AUTHOR:  Kratovi4
VERSION : 2.0
STRUCT
DRV: ARRAY  [1 .. 35] OF
"DRV"; // Array
END_STRUCT ;
BEGIN
END_DATA_BLOCK


DATA_BLOCK DB304
TITLE =Valves
AUTHOR:  Kratovi4
VERSION : 2.0
STRUCT
DRV: ARRAY  [1 .. 10] OF
"DRV"; // Array
END_STRUCT ;
BEGIN
END_DATA_BLOCK


DATA_BLOCK DB314
TITLE =Valves
AUTHOR:  Kratovi4
VERSION : 2.0
STRUCT
DRV: ARRAY  [1 .. 10] OF
"DRV"; // Array
END_STRUCT ;
BEGIN
END_DATA_BLOCK


DATA_BLOCK DB324
TITLE =Valves
AUTHOR:  Kratovi4
VERSION : 2.0
STRUCT
DRV: ARRAY  [1 .. 10] OF
"DRV"; // Array
END_STRUCT ;
BEGIN
END_DATA_BLOCK


DATA_BLOCK DB344
TITLE =Valves
AUTHOR:  Kratovi4
VERSION : 2.0
STRUCT
DRV: ARRAY  [1 .. 10] OF
"DRV"; // Array
END_STRUCT ;
BEGIN
END_DATA_BLOCK


DATA_BLOCK DB354
TITLE =Valves
AUTHOR:  Kratovi4
VERSION : 2.0
STRUCT
DRV: ARRAY  [1 .. 5] OF
"DRV"; // Array
END_STRUCT ;
BEGIN
END_DATA_BLOCK


DATA_BLOCK DB434
TITLE =Valves
AUTHOR:  Kratovi4
VERSION : 2.0
STRUCT
DRV: ARRAY  [1 .. 30] OF
"DRV"; // Array
END_STRUCT ;
BEGIN
END_DATA_BLOCK


DATA_BLOCK DB444
TITLE =Valves
AUTHOR:  Kratovi4
VERSION : 2.0
STRUCT
DRV: ARRAY  [1 .. 10] OF
"DRV"; // Array
END_STRUCT ;
BEGIN
END_DATA_BLOCK


DATA_BLOCK DB454
TITLE =Valves
AUTHOR:  Kratovi4
VERSION : 2.0
STRUCT
DRV: ARRAY  [1 .. 10] OF
"DRV"; // Array
END_STRUCT ;
BEGIN
END_DATA_BLOCK


DATA_BLOCK DB464
TITLE =Valves
AUTHOR:  Kratovi4
VERSION : 2.0
STRUCT
DRV: ARRAY  [1 .. 10] OF
"DRV"; // Array
END_STRUCT ;
BEGIN
END_DATA_BLOCK


DATA_BLOCK DB474
TITLE =Valves
AUTHOR:  Kratovi4
VERSION : 2.0
STRUCT
DRV: ARRAY  [1 .. 10] OF
"DRV"; // Array
END_STRUCT ;
BEGIN
END_DATA_BLOCK


DATA_BLOCK DB494
TITLE =Valves
AUTHOR:  Kratovi4
VERSION : 2.0
STRUCT
DRV: ARRAY  [1 .. 5] OF
"DRV"; // Array
END_STRUCT ;
BEGIN
END_DATA_BLOCK


DATA_BLOCK DB514
TITLE =Valves
AUTHOR:  Kratovi4
VERSION : 2.0
STRUCT
DRV: ARRAY  [1 .. 5] OF
"DRV"; // Array
END_STRUCT ;
BEGIN
END_DATA_BLOCK


DATA_BLOCK DB524
TITLE =Valves
AUTHOR:  Kratovi4
VERSION : 2.0
STRUCT
DRV: ARRAY  [1 .. 5] OF
"DRV"; // Array
END_STRUCT ;
BEGIN
END_DATA_BLOCK


DATA_BLOCK DB534
TITLE =Valves
AUTHOR:  Kratovi4
VERSION : 2.0
STRUCT
DRV: ARRAY  [1 .. 5] OF
"DRV"; // Array
END_STRUCT ;
BEGIN
END_DATA_BLOCK


DATA_BLOCK DB544
TITLE =Valves
AUTHOR:  Kratovi4
VERSION : 2.0
STRUCT
DRV: ARRAY  [1 .. 10] OF
"DRV"; // Array
END_STRUCT ;
BEGIN
END_DATA_BLOCK


DATA_BLOCK DB554
TITLE =Valves
AUTHOR:  Kratovi4
VERSION : 2.0
STRUCT
DRV: ARRAY  [1 .. 5] OF
"DRV"; // Array
END_STRUCT ;
BEGIN
END_DATA_BLOCK


DATA_BLOCK DB564
TITLE =Valves
AUTHOR:  Kratovi4
VERSION : 2.0
STRUCT
DRV: ARRAY  [1 .. 15] OF
"DRV"; // Array
END_STRUCT ;
BEGIN
END_DATA_BLOCK


DATA_BLOCK DB574
TITLE =Valves
AUTHOR:  Kratovi4
VERSION : 2.0
STRUCT
DRV: ARRAY  [1 .. 15] OF
"DRV"; // Array
END_STRUCT ;
BEGIN
END_DATA_BLOCK


DATA_BLOCK DB584
TITLE =Valves
AUTHOR:  Kratovi4
VERSION : 2.0
STRUCT
DRV: ARRAY  [1 .. 15] OF
"DRV"; // Array
END_STRUCT ;
BEGIN
END_DATA_BLOCK


DATA_BLOCK DB604
TITLE =Valves
AUTHOR:  Kratovi4
VERSION : 2.0
STRUCT
DRV: ARRAY  [1 .. 25] OF
"DRV"; // Array
END_STRUCT ;
BEGIN
END_DATA_BLOCK


DATA_BLOCK DB614
TITLE =Valves
AUTHOR:  Kratovi4
VERSION : 2.0
STRUCT
DRV: ARRAY  [1 .. 5] OF
"DRV"; // Array
END_STRUCT ;
BEGIN
END_DATA_BLOCK


DATA_BLOCK DB624
TITLE =Valves
AUTHOR:  Kratovi4
VERSION : 2.0
STRUCT
DRV: ARRAY  [1 .. 5] OF
"DRV"; // Array
END_STRUCT ;
BEGIN
END_DATA_BLOCK


DATA_BLOCK DB634
TITLE =Valves
AUTHOR:  Kratovi4
VERSION : 2.0
STRUCT
DRV: ARRAY  [1 .. 5] OF
"DRV"; // Array
END_STRUCT ;
BEGIN
END_DATA_BLOCK


DATA_BLOCK DB644
TITLE =Valves
AUTHOR:  Kratovi4
VERSION : 2.0
STRUCT
DRV: ARRAY  [1 .. 5] OF
"DRV"; // Array
END_STRUCT ;
BEGIN
END_DATA_BLOCK


DATA_BLOCK DB674
TITLE =Valves
AUTHOR:  Kratovi4
VERSION : 2.0
STRUCT
DRV: ARRAY  [1 .. 10] OF
"DRV"; // Array
END_STRUCT ;
BEGIN
END_DATA_BLOCK


DATA_BLOCK DB684
TITLE =Valves
AUTHOR:  Kratovi4
VERSION : 2.0
STRUCT
DRV: ARRAY  [1 .. 5] OF
"DRV"; // Array
END_STRUCT ;
BEGIN
END_DATA_BLOCK


DATA_BLOCK DB694
TITLE =Valves
AUTHOR:  Kratovi4
VERSION : 2.0
STRUCT
DRV: ARRAY  [1 .. 5] OF
"DRV"; // Array
END_STRUCT ;
BEGIN
END_DATA_BLOCK


DATA_BLOCK DB704
TITLE =Valves
AUTHOR:  Kratovi4
VERSION : 2.0
STRUCT
DRV: ARRAY  [1 .. 5] OF
"DRV"; // Array
END_STRUCT ;
BEGIN
END_DATA_BLOCK


DATA_BLOCK DB714
TITLE =Valves
AUTHOR:  Kratovi4
VERSION : 2.0
STRUCT
DRV: ARRAY  [1 .. 5] OF
"DRV"; // Array
END_STRUCT ;
BEGIN
END_DATA_BLOCK


DATA_BLOCK DB724
TITLE =Valves
AUTHOR:  Kratovi4
VERSION : 2.0
STRUCT
DRV: ARRAY  [1 .. 25] OF
"DRV"; // Array
END_STRUCT ;
BEGIN
END_DATA_BLOCK


DATA_BLOCK DB734
TITLE =Valves
AUTHOR:  Kratovi4
VERSION : 2.0
STRUCT
DRV: ARRAY  [1 .. 5] OF
"DRV"; // Array
END_STRUCT ;
BEGIN
END_DATA_BLOCK


DATA_BLOCK DB744
TITLE =Valves
AUTHOR:  Kratovi4
VERSION : 2.0
STRUCT
DRV: ARRAY  [1 .. 5] OF
"DRV"; // Array
END_STRUCT ;
BEGIN
END_DATA_BLOCK


DATA_BLOCK DB754
TITLE =Valves
AUTHOR:  Kratovi4
VERSION : 2.0
STRUCT
DRV: ARRAY  [1 .. 5] OF
"DRV"; // Array
END_STRUCT ;
BEGIN
END_DATA_BLOCK


DATA_BLOCK DB774
TITLE =Valves
AUTHOR:  Kratovi4
VERSION : 2.0
STRUCT
DRV: ARRAY  [1 .. 10] OF
"DRV"; // Array
END_STRUCT ;
BEGIN
END_DATA_BLOCK


DATA_BLOCK DB784
TITLE =Valves
AUTHOR:  Kratovi4
VERSION : 2.0
STRUCT
DRV: ARRAY  [1 .. 5] OF
"DRV"; // Array
END_STRUCT ;
BEGIN
END_DATA_BLOCK


DATA_BLOCK DB794
TITLE =Valves
AUTHOR:  Kratovi4
VERSION : 2.0
STRUCT
DRV: ARRAY  [1 .. 10] OF
"DRV"; // Array
END_STRUCT ;
BEGIN
END_DATA_BLOCK


DATA_BLOCK DB804
TITLE =Valves
AUTHOR:  Kratovi4
VERSION : 2.0
STRUCT
DRV: ARRAY  [1 .. 10] OF
"DRV"; // Array
END_STRUCT ;
BEGIN
END_DATA_BLOCK


DATA_BLOCK DB814
TITLE =Valves
AUTHOR:  Kratovi4
VERSION : 2.0
STRUCT
DRV: ARRAY  [1 .. 10] OF
"DRV"; // Array
END_STRUCT ;
BEGIN
END_DATA_BLOCK


DATA_BLOCK DB834
TITLE =Valves
AUTHOR:  Kratovi4
VERSION : 2.0
STRUCT
DRV: ARRAY  [1 .. 5] OF
"DRV"; // Array
END_STRUCT ;
BEGIN
END_DATA_BLOCK


DATA_BLOCK DB844
TITLE =Valves
AUTHOR:  Kratovi4
VERSION : 2.0
STRUCT
DRV: ARRAY  [1 .. 5] OF
"DRV"; // Array
END_STRUCT ;
BEGIN
END_DATA_BLOCK


DATA_BLOCK DB854
TITLE =Valves
AUTHOR:  Kratovi4
VERSION : 2.0
STRUCT
DRV: ARRAY  [1 .. 10] OF
"DRV"; // Array
END_STRUCT ;
BEGIN
END_DATA_BLOCK


DATA_BLOCK DB864
TITLE =Valves
AUTHOR:  Kratovi4
VERSION : 2.0
STRUCT
DRV: ARRAY  [1 .. 10] OF
"DRV"; // Array
END_STRUCT ;
BEGIN
END_DATA_BLOCK


DATA_BLOCK DB884
TITLE =Valves
AUTHOR:  Kratovi4
VERSION : 2.0
STRUCT
DRV: ARRAY  [1 .. 10] OF
"DRV"; // Array
END_STRUCT ;
BEGIN
END_DATA_BLOCK


DATA_BLOCK DB115
TITLE =Pumps
AUTHOR:  Kratovi4
VERSION : 2.0
STRUCT
DRV: ARRAY  [1 .. 5] OF
"DRV"; // Array
END_STRUCT ;
BEGIN
END_DATA_BLOCK


DATA_BLOCK DB125
TITLE =Pumps
AUTHOR:  Kratovi4
VERSION : 2.0
STRUCT
DRV: ARRAY  [1 .. 5] OF
"DRV"; // Array
END_STRUCT ;
BEGIN
END_DATA_BLOCK


DATA_BLOCK DB145
TITLE =Pumps
AUTHOR:  Kratovi4
VERSION : 2.0
STRUCT
DRV: ARRAY  [1 .. 5] OF
"DRV"; // Array
END_STRUCT ;
BEGIN
END_DATA_BLOCK


DATA_BLOCK DB165
TITLE =Pumps
AUTHOR:  Kratovi4
VERSION : 2.0
STRUCT
DRV: ARRAY  [1 .. 5] OF
"DRV"; // Array
END_STRUCT ;
BEGIN
END_DATA_BLOCK


DATA_BLOCK DB175
TITLE =Pumps
AUTHOR:  Kratovi4
VERSION : 2.0
STRUCT
DRV: ARRAY  [1 .. 5] OF
"DRV"; // Array
END_STRUCT ;
BEGIN
END_DATA_BLOCK


DATA_BLOCK DB215
TITLE =Pumps
AUTHOR:  Kratovi4
VERSION : 2.0
STRUCT
DRV: ARRAY  [1 .. 5] OF
"DRV"; // Array
END_STRUCT ;
BEGIN
END_DATA_BLOCK


DATA_BLOCK DB225
TITLE =Pumps
AUTHOR:  Kratovi4
VERSION : 2.0
STRUCT
DRV: ARRAY  [1 .. 5] OF
"DRV"; // Array
END_STRUCT ;
BEGIN
END_DATA_BLOCK


DATA_BLOCK DB235
TITLE =Pumps
AUTHOR:  Kratovi4
VERSION : 2.0
STRUCT
DRV: ARRAY  [1 .. 5] OF
"DRV"; // Array
END_STRUCT ;
BEGIN
END_DATA_BLOCK


DATA_BLOCK DB245
TITLE =Pumps
AUTHOR:  Kratovi4
VERSION : 2.0
STRUCT
DRV: ARRAY  [1 .. 15] OF
"DRV"; // Array
END_STRUCT ;
BEGIN
END_DATA_BLOCK


DATA_BLOCK DB255
TITLE =Pumps
AUTHOR:  Kratovi4
VERSION : 2.0
STRUCT
DRV: ARRAY  [1 .. 15] OF
"DRV"; // Array
END_STRUCT ;
BEGIN
END_DATA_BLOCK


DATA_BLOCK DB265
TITLE =Pumps
AUTHOR:  Kratovi4
VERSION : 2.0
STRUCT
DRV: ARRAY  [1 .. 15] OF
"DRV"; // Array
END_STRUCT ;
BEGIN
END_DATA_BLOCK


DATA_BLOCK DB285
TITLE =Pumps
AUTHOR:  Kratovi4
VERSION : 2.0
STRUCT
DRV: ARRAY  [1 .. 5] OF
"DRV"; // Array
END_STRUCT ;
BEGIN
END_DATA_BLOCK


DATA_BLOCK DB295
TITLE =Pumps
AUTHOR:  Kratovi4
VERSION : 2.0
STRUCT
DRV: ARRAY  [1 .. 10] OF
"DRV"; // Array
END_STRUCT ;
BEGIN
END_DATA_BLOCK


DATA_BLOCK DB305
TITLE =Pumps
AUTHOR:  Kratovi4
VERSION : 2.0
STRUCT
DRV: ARRAY  [1 .. 5] OF
"DRV"; // Array
END_STRUCT ;
BEGIN
END_DATA_BLOCK


DATA_BLOCK DB315
TITLE =Pumps
AUTHOR:  Kratovi4
VERSION : 2.0
STRUCT
DRV: ARRAY  [1 .. 5] OF
"DRV"; // Array
END_STRUCT ;
BEGIN
END_DATA_BLOCK


DATA_BLOCK DB325
TITLE =Pumps
AUTHOR:  Kratovi4
VERSION : 2.0
STRUCT
DRV: ARRAY  [1 .. 5] OF
"DRV"; // Array
END_STRUCT ;
BEGIN
END_DATA_BLOCK


DATA_BLOCK DB345
TITLE =Pumps
AUTHOR:  Kratovi4
VERSION : 2.0
STRUCT
DRV: ARRAY  [1 .. 5] OF
"DRV"; // Array
END_STRUCT ;
BEGIN
END_DATA_BLOCK


DATA_BLOCK DB435
TITLE =Pumps
AUTHOR:  Kratovi4
VERSION : 2.0
STRUCT
DRV: ARRAY  [1 .. 5] OF
"DRV"; // Array
END_STRUCT ;
BEGIN
END_DATA_BLOCK


DATA_BLOCK DB445
TITLE =Pumps
AUTHOR:  Kratovi4
VERSION : 2.0
STRUCT
DRV: ARRAY  [1 .. 15] OF
"DRV"; // Array
END_STRUCT ;
BEGIN
END_DATA_BLOCK


DATA_BLOCK DB455
TITLE =Pumps
AUTHOR:  Kratovi4
VERSION : 2.0
STRUCT
DRV: ARRAY  [1 .. 15] OF
"DRV"; // Array
END_STRUCT ;
BEGIN
END_DATA_BLOCK


DATA_BLOCK DB465
TITLE =Pumps
AUTHOR:  Kratovi4
VERSION : 2.0
STRUCT
DRV: ARRAY  [1 .. 15] OF
"DRV"; // Array
END_STRUCT ;
BEGIN
END_DATA_BLOCK


DATA_BLOCK DB475
TITLE =Pumps
AUTHOR:  Kratovi4
VERSION : 2.0
STRUCT
DRV: ARRAY  [1 .. 15] OF
"DRV"; // Array
END_STRUCT ;
BEGIN
END_DATA_BLOCK


DATA_BLOCK DB495
TITLE =Pumps
AUTHOR:  Kratovi4
VERSION : 2.0
STRUCT
DRV: ARRAY  [1 .. 5] OF
"DRV"; // Array
END_STRUCT ;
BEGIN
END_DATA_BLOCK


DATA_BLOCK DB545
TITLE =Pumps
AUTHOR:  Kratovi4
VERSION : 2.0
STRUCT
DRV: ARRAY  [1 .. 5] OF
"DRV"; // Array
END_STRUCT ;
BEGIN
END_DATA_BLOCK


DATA_BLOCK DB555
TITLE =Pumps
AUTHOR:  Kratovi4
VERSION : 2.0
STRUCT
DRV: ARRAY  [1 .. 5] OF
"DRV"; // Array
END_STRUCT ;
BEGIN
END_DATA_BLOCK


DATA_BLOCK DB565
TITLE =Pumps
AUTHOR:  Kratovi4
VERSION : 2.0
STRUCT
DRV: ARRAY  [1 .. 5] OF
"DRV"; // Array
END_STRUCT ;
BEGIN
END_DATA_BLOCK


DATA_BLOCK DB575
TITLE =Pumps
AUTHOR:  Kratovi4
VERSION : 2.0
STRUCT
DRV: ARRAY  [1 .. 5] OF
"DRV"; // Array
END_STRUCT ;
BEGIN
END_DATA_BLOCK


DATA_BLOCK DB585
TITLE =Pumps
AUTHOR:  Kratovi4
VERSION : 2.0
STRUCT
DRV: ARRAY  [1 .. 5] OF
"DRV"; // Array
END_STRUCT ;
BEGIN
END_DATA_BLOCK


DATA_BLOCK DB605
TITLE =Pumps
AUTHOR:  Kratovi4
VERSION : 2.0
STRUCT
DRV: ARRAY  [1 .. 5] OF
"DRV"; // Array
END_STRUCT ;
BEGIN
END_DATA_BLOCK


DATA_BLOCK DB625
TITLE =Pumps
AUTHOR:  Kratovi4
VERSION : 2.0
STRUCT
DRV: ARRAY  [1 .. 5] OF
"DRV"; // Array
END_STRUCT ;
BEGIN
END_DATA_BLOCK


DATA_BLOCK DB635
TITLE =Pumps
AUTHOR:  Kratovi4
VERSION : 2.0
STRUCT
DRV: ARRAY  [1 .. 5] OF
"DRV"; // Array
END_STRUCT ;
BEGIN
END_DATA_BLOCK


DATA_BLOCK DB645
TITLE =Pumps
AUTHOR:  Kratovi4
VERSION : 2.0
STRUCT
DRV: ARRAY  [1 .. 5] OF
"DRV"; // Array
END_STRUCT ;
BEGIN
END_DATA_BLOCK


DATA_BLOCK DB675
TITLE =Pumps
AUTHOR:  Kratovi4
VERSION : 2.0
STRUCT
DRV: ARRAY  [1 .. 5] OF
"DRV"; // Array
END_STRUCT ;
BEGIN
END_DATA_BLOCK


DATA_BLOCK DB685
TITLE =Pumps
AUTHOR:  Kratovi4
VERSION : 2.0
STRUCT
DRV: ARRAY  [1 .. 15] OF
"DRV"; // Array
END_STRUCT ;
BEGIN
END_DATA_BLOCK


DATA_BLOCK DB695
TITLE =Pumps
AUTHOR:  Kratovi4
VERSION : 2.0
STRUCT
DRV: ARRAY  [1 .. 15] OF
"DRV"; // Array
END_STRUCT ;
BEGIN
END_DATA_BLOCK


DATA_BLOCK DB705
TITLE =Pumps
AUTHOR:  Kratovi4
VERSION : 2.0
STRUCT
DRV: ARRAY  [1 .. 15] OF
"DRV"; // Array
END_STRUCT ;
BEGIN
END_DATA_BLOCK


DATA_BLOCK DB715
TITLE =Pumps
AUTHOR:  Kratovi4
VERSION : 2.0
STRUCT
DRV: ARRAY  [1 .. 15] OF
"DRV"; // Array
END_STRUCT ;
BEGIN
END_DATA_BLOCK


DATA_BLOCK DB725
TITLE =Pumps
AUTHOR:  Kratovi4
VERSION : 2.0
STRUCT
DRV: ARRAY  [1 .. 5] OF
"DRV"; // Array
END_STRUCT ;
BEGIN
END_DATA_BLOCK


DATA_BLOCK DB735
TITLE =Pumps
AUTHOR:  Kratovi4
VERSION : 2.0
STRUCT
DRV: ARRAY  [1 .. 15] OF
"DRV"; // Array
END_STRUCT ;
BEGIN
END_DATA_BLOCK


DATA_BLOCK DB745
TITLE =Pumps
AUTHOR:  Kratovi4
VERSION : 2.0
STRUCT
DRV: ARRAY  [1 .. 15] OF
"DRV"; // Array
END_STRUCT ;
BEGIN
END_DATA_BLOCK


DATA_BLOCK DB755
TITLE =Pumps
AUTHOR:  Kratovi4
VERSION : 2.0
STRUCT
DRV: ARRAY  [1 .. 15] OF
"DRV"; // Array
END_STRUCT ;
BEGIN
END_DATA_BLOCK


DATA_BLOCK DB775
TITLE =Pumps
AUTHOR:  Kratovi4
VERSION : 2.0
STRUCT
DRV: ARRAY  [1 .. 5] OF
"DRV"; // Array
END_STRUCT ;
BEGIN
END_DATA_BLOCK


DATA_BLOCK DB785
TITLE =Pumps
AUTHOR:  Kratovi4
VERSION : 2.0
STRUCT
DRV: ARRAY  [1 .. 5] OF
"DRV"; // Array
END_STRUCT ;
BEGIN
END_DATA_BLOCK


DATA_BLOCK DB795
TITLE =Pumps
AUTHOR:  Kratovi4
VERSION : 2.0
STRUCT
DRV: ARRAY  [1 .. 5] OF
"DRV"; // Array
END_STRUCT ;
BEGIN
END_DATA_BLOCK


DATA_BLOCK DB805
TITLE =Pumps
AUTHOR:  Kratovi4
VERSION : 2.0
STRUCT
DRV: ARRAY  [1 .. 5] OF
"DRV"; // Array
END_STRUCT ;
BEGIN
END_DATA_BLOCK


DATA_BLOCK DB815
TITLE =Pumps
AUTHOR:  Kratovi4
VERSION : 2.0
STRUCT
DRV: ARRAY  [1 .. 5] OF
"DRV"; // Array
END_STRUCT ;
BEGIN
END_DATA_BLOCK


DATA_BLOCK DB835
TITLE =Pumps
AUTHOR:  Kratovi4
VERSION : 2.0
STRUCT
DRV: ARRAY  [1 .. 15] OF
"DRV"; // Array
END_STRUCT ;
BEGIN
END_DATA_BLOCK


DATA_BLOCK DB845
TITLE =Pumps
AUTHOR:  Kratovi4
VERSION : 2.0
STRUCT
DRV: ARRAY  [1 .. 15] OF
"DRV"; // Array
END_STRUCT ;
BEGIN
END_DATA_BLOCK


DATA_BLOCK DB855
TITLE =Pumps
AUTHOR:  Kratovi4
VERSION : 2.0
STRUCT
DRV: ARRAY  [1 .. 15] OF
"DRV"; // Array
END_STRUCT ;
BEGIN
END_DATA_BLOCK


DATA_BLOCK DB865
TITLE =Pumps
AUTHOR:  Kratovi4
VERSION : 2.0
STRUCT
DRV: ARRAY  [1 .. 5] OF
"DRV"; // Array
END_STRUCT ;
BEGIN
END_DATA_BLOCK


DATA_BLOCK DB885
TITLE =Pumps
AUTHOR:  Kratovi4
VERSION : 2.0
STRUCT
DRV: ARRAY  [1 .. 5] OF
"DRV"; // Array
END_STRUCT ;
BEGIN
END_DATA_BLOCK


DATA_BLOCK DB567
TITLE =Cheese Mixers
AUTHOR:  Kratovi4
VERSION : 2.0
STRUCT
MXR: ARRAY  [1 .. 5] OF
"MXR_CM"; // Array
END_STRUCT ;
BEGIN
END_DATA_BLOCK


DATA_BLOCK DB577
TITLE =Cheese Mixers
AUTHOR:  Kratovi4
VERSION : 2.0
STRUCT
MXR: ARRAY  [1 .. 5] OF
"MXR_CM"; // Array
END_STRUCT ;
BEGIN
END_DATA_BLOCK


DATA_BLOCK DB587
TITLE =Cheese Mixers
AUTHOR:  Kratovi4
VERSION : 2.0
STRUCT
MXR: ARRAY  [1 .. 5] OF
"MXR_CM"; // Array
END_STRUCT ;
BEGIN
END_DATA_BLOCK


DATA_BLOCK DB119
TITLE =Counters
AUTHOR:  Kratovi4
VERSION : 2.0
STRUCT
SNC: ARRAY  [1 .. 5] OF
"SNC"; // Array
END_STRUCT ;
BEGIN
END_DATA_BLOCK


DATA_BLOCK DB129
TITLE =Counters
AUTHOR:  Kratovi4
VERSION : 2.0
STRUCT
SNC: ARRAY  [1 .. 5] OF
"SNC"; // Array
END_STRUCT ;
BEGIN
END_DATA_BLOCK


DATA_BLOCK DB219
TITLE =Counters
AUTHOR:  Kratovi4
VERSION : 2.0
STRUCT
SNC: ARRAY  [1 .. 5] OF
"SNC"; // Array
END_STRUCT ;
BEGIN
END_DATA_BLOCK


DATA_BLOCK DB229
TITLE =Counters
AUTHOR:  Kratovi4
VERSION : 2.0
STRUCT
SNC: ARRAY  [1 .. 5] OF
"SNC"; // Array
END_STRUCT ;
BEGIN
END_DATA_BLOCK


DATA_BLOCK DB239
TITLE =Counters
AUTHOR:  Kratovi4
VERSION : 2.0
STRUCT
SNC: ARRAY  [1 .. 5] OF
"SNC"; // Array
END_STRUCT ;
BEGIN
END_DATA_BLOCK


DATA_BLOCK DB299
TITLE =Counters
AUTHOR:  Kratovi4
VERSION : 2.0
STRUCT
SNC: ARRAY  [1 .. 10] OF
"SNC"; // Array
END_STRUCT ;
BEGIN
END_DATA_BLOCK


DATA_BLOCK DB439
TITLE =Counters
AUTHOR:  Kratovi4
VERSION : 2.0
STRUCT
SNC: ARRAY  [1 .. 10] OF
"SNC"; // Array
END_STRUCT ;
BEGIN
END_DATA_BLOCK


DATA_BLOCK DB519
TITLE =Counters
AUTHOR:  Kratovi4
VERSION : 2.0
STRUCT
SNC: ARRAY  [1 .. 5] OF
"SNC"; // Array
END_STRUCT ;
BEGIN
END_DATA_BLOCK


DATA_BLOCK DB549
TITLE =Counters
AUTHOR:  Kratovi4
VERSION : 2.0
STRUCT
SNC: ARRAY  [1 .. 5] OF
"SNC"; // Array
END_STRUCT ;
BEGIN
END_DATA_BLOCK


DATA_BLOCK DB679
TITLE =Counters
AUTHOR:  Kratovi4
VERSION : 2.0
STRUCT
SNC: ARRAY  [1 .. 5] OF
"SNC"; // Array
END_STRUCT ;
BEGIN
END_DATA_BLOCK


DATA_BLOCK DB729
TITLE =Counters
AUTHOR:  Kratovi4
VERSION : 2.0
STRUCT
SNC: ARRAY  [1 .. 5] OF
"SNC"; // Array
END_STRUCT ;
BEGIN
END_DATA_BLOCK


DATA_BLOCK DB779
TITLE =Counters
AUTHOR:  Kratovi4
VERSION : 2.0
STRUCT
SNC: ARRAY  [1 .. 5] OF
"SNC"; // Array
END_STRUCT ;
BEGIN
END_DATA_BLOCK


DATA_BLOCK DB99
TITLE =Setpoint
AUTHOR:  Kratovi4
VERSION : 2.0
STRUCT
SC: ARRAY  [1 .. 5] OF
"SC"; // Array
END_STRUCT ;
BEGIN
END_DATA_BLOCK


